{attribute 'qualified_only'}
VAR_GLOBAL

END_VAR

(* stored: Version 1.1.0.1, ProductVersion 3.1.4024.12
   GVL GVL_Main: Id {13c37659-0099-44ae-90c0-9ff26dea58a3} *)
